TYPE DS_VisuElement :
STRUCT
	CurrentUserGroupId 	: int;
	CurrentUserName		: WSTRING;
	CurrentVisu			: STRING;

	
END_STRUCT
END_TYPE

(* stored: Version 1.1.0.1, ProductVersion 3.1.4024.12
   DUT DS_VisuElement: Id {009de7ef-0826-4c72-840e-3aa11b5e58b5} *)
